Omron CX-Programmer project 新工程 (CX-Programmer 9.51)

# PLC officeLight: CP1E N30

## Global symbols (name address type ; comment)
0.00 BOOL  ; 启动
0.01 BOOL  ; 停止
0.02 BOOL  ; 手动开关
0.03 BOOL  ; 道路1
1 CHANNEL  ; 1秒脉冲
100.00 BOOL  ; 红灯1
100.01 BOOL  ; 黄灯1
100.02 BOOL  ; 绿灯1
100.03 BOOL  ; 红灯1
100.04 BOOL  ; 红灯2
100.05 BOOL  ; 黄灯2
100.06 BOOL  ; 绿灯2
200.00 BOOL  ; 启动保持
20.00 BOOL  ; 手动
30.00 BOOL  ; 道路1
30.01 BOOL  ; 启动保持
T000 BOOL  ; 绿1
T001 BOOL  ; 闪烁1
T002 BOOL  ; 黄1
T003 BOOL  ; 绿2
T004 BOOL  ; 闪烁2
T005 BOOL  ; 黄2
启动开关（自动） 0.00 BOOL  ; 启动开关

## Program 新程序1 (cyclic task 0)

### Section 段1

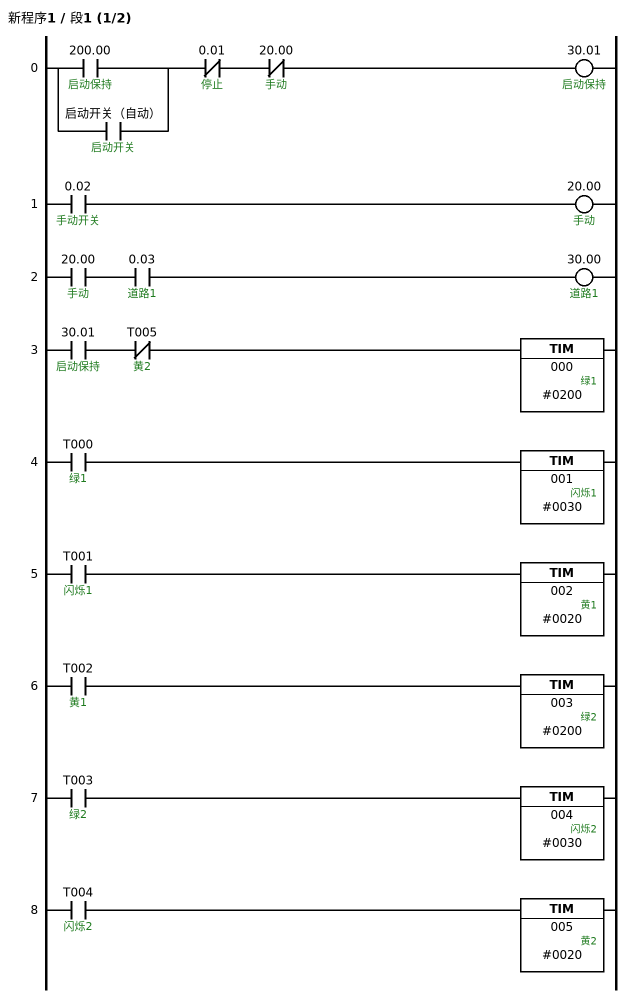
; rung 0
LD 200.00  ; 启动保持
OR 启动开关（自动）  ; 启动开关
ANDNOT 0.01  ; 停止
ANDNOT 20.00  ; 手动
OUT 30.01  ; 启动保持
; rung 1
LD 0.02  ; 手动开关
OUT 20.00  ; 手动
; rung 2
LD 20.00  ; 手动
AND 0.03  ; 道路1
OUT 30.00  ; 道路1
; rung 3
LD 30.01  ; 启动保持
ANDNOT T005  ; 黄2
TIM 000 #0200  ; 绿1
; rung 4
LD T000  ; 绿1
TIM 001 #0030  ; 闪烁1
; rung 5
LD T001  ; 闪烁1
TIM 002 #0020  ; 黄1
; rung 6
LD T002  ; 黄1
TIM 003 #0200  ; 绿2
; rung 7
LD T003  ; 绿2
TIM 004 #0030  ; 闪烁2
; rung 8
LD T004  ; 闪烁2
TIM 005 #0020  ; 黄2

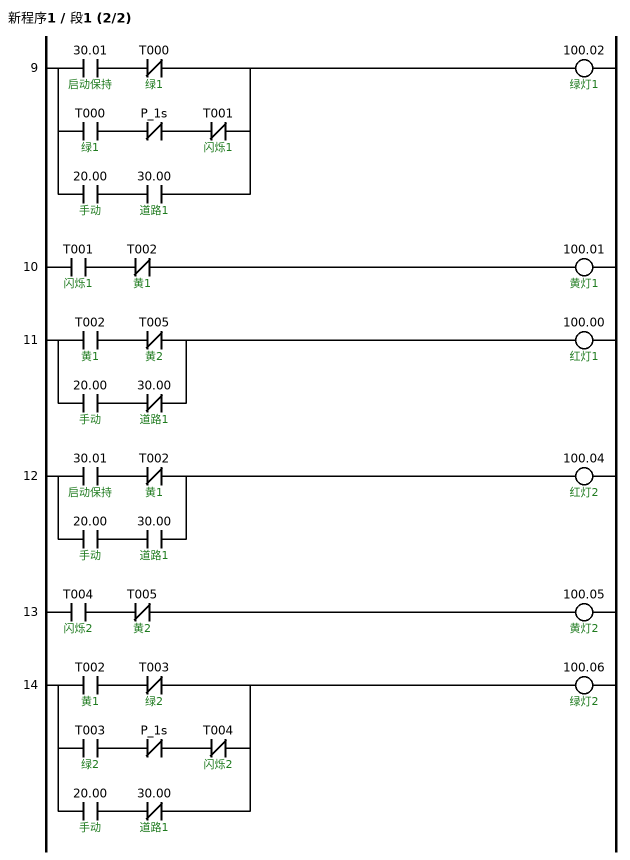
; rung 9
LD 30.01  ; 启动保持
ANDNOT T000  ; 绿1
LD T000  ; 绿1
ANDNOT P_1s
ANDNOT T001  ; 闪烁1
ORLD
LD 20.00  ; 手动
AND 30.00  ; 道路1
ORLD
OUT 100.02  ; 绿灯1
; rung 10
LD T001  ; 闪烁1
ANDNOT T002  ; 黄1
OUT 100.01  ; 黄灯1
; rung 11
LD T002  ; 黄1
ANDNOT T005  ; 黄2
LD 20.00  ; 手动
ANDNOT 30.00  ; 道路1
ORLD
OUT 100.00  ; 红灯1
; rung 12
LD 30.01  ; 启动保持
ANDNOT T002  ; 黄1
LD 20.00  ; 手动
AND 30.00  ; 道路1
ORLD
OUT 100.04  ; 红灯2
; rung 13
LD T004  ; 闪烁2
ANDNOT T005  ; 黄2
OUT 100.05  ; 黄灯2
; rung 14
LD T002  ; 黄1
ANDNOT T003  ; 绿2
LD T003  ; 绿2
ANDNOT P_1s
ANDNOT T004  ; 闪烁2
ORLD
LD 20.00  ; 手动
ANDNOT 30.00  ; 道路1
ORLD
OUT 100.06  ; 绿灯2
; rung 15
END(001)

### Section END
; rung 0
END(001)